FUNCTION_BLOCK PUBLIC FB_DecoratorTomato EXTENDS FB_Decorator
VAR_INPUT
END_VAR
VAR_OUTPUT
END_VAR
VAR
	bWholefood		: BOOL;
END_VAR

PROPERTY PUBLIC bWholefoodProduct : BOOL
GET
bWholefoodProduct := THIS^.bWholefood;
END_GET
SET
THIS^.bWholefood := bWholefoodProduct;
END_SET
END_PROPERTY

METHOD FB_init : BOOL
VAR_INPUT
	bInitRetains		: BOOL; // if TRUE, the retain variables are initialized (warm start / cold start)
	bInCopyCode			: BOOL;  // if TRUE, the instance afterwards gets moved into the copy code (online change)
	ipSideOrder			: I_Pizza;
	bWholefoodProduct	: BOOL;
END_VAR
THIS^.bWholefood := bWholefoodProduct;
END_METHOD

METHOD GetDescription : STRING
IF (SUPER^.ipSideOrder <> 0) THEN
	GetDescription := CONCAT (SUPER^.ipSideOrder.GetDescription(), ' - Tomato');
	IF (THIS^.bWholefoodProduct) THEN
	GetDescription := CONCAT (GetDescription, ' (WholefoodProduct) ');
	END_IF
END_IF
END_METHOD

METHOD GetPrice : LREAL
IF (SUPER^.ipSideOrder <> 0) THEN
	GetPrice := SUPER^.ipSideOrder.GetPrice() + 0.9;
	IF (THIS^.bWholefood) THEN
		GetPrice := GetPrice + 0.3;
	END_IF
END_IF
END_METHOD

END_FUNCTION_BLOCK

(* stored: Version 1.1.0.1, ProductVersion 3.1.4022.16
   POU FB_DecoratorTomato: Id {6a23dffc-d9d0-4e5c-bc48-3acf097e19de}, SpecialFunc None
   Property bWholefoodProduct: Id {65856119-ca3c-4762-90bd-46b97fff58cd}
   Get Get: Id {c62384ce-341e-41f3-b682-5c77937f6e2b}
   Set Set: Id {80b4dbd7-5926-49ed-8080-9fa8569131ce}
   Method FB_init: Id {e7580572-2915-4701-a566-ac200c74698f}
   Method GetDescription: Id {56e36320-0678-448c-833e-b8dbe091013a}
   Method GetPrice: Id {7a4344c4-2641-474b-9a89-327e457a43d6} *)
